// Mitsubishi GX Works2 project: exercicio 4   PLC: Q03UDV

PROGRAM MAIN
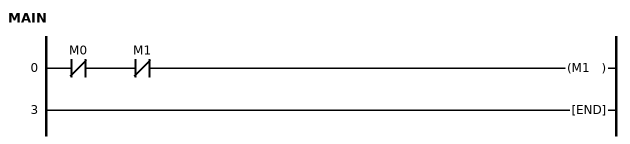
0     LDI     M0
      ANI     M1
      OUT     M1
3     END
END_PROGRAM
